TYPE Rec_Compress :
	STRUCT
		Initial_Speed				:LREAL;
		Initial_Distance			:LREAL;
		Shield_Dwell				:LREAL;
		Relax_Distance				:LREAL;
		Retract_Speed				:LREAL;
	END_STRUCT
END_TYPE

(* stored: Version 1.1.0.1, ProductVersion 3.1.4020.12
   DUT Rec_Compress: Id {ebb9e94e-f8ca-41b2-9119-d21a16b1d90d} *)
